(* Logix 5000 project; controller VET 1756-L62 rev 19.52; software revision 19.01; part 23 of 27 *)
(* tags used below, declared in another part *)
   Aux : DINT[500];
   Eqp : Equipo[50];
   I : Index;
   PID : PID_Struct;
   RunHours : DINT[1000];
   RunSegs : DINT[1000];
   RunStarts : DINT[1000];
   _Eqp : Equipo[800];
   _Eqp_Cfg : Eqp_Cfg[800];
   _SS : Soft_Starter[20];
   _Typlgie : Eqp_Typologie[800];   // Process Flow Typologie
   borrar : DINT[100];
   comandos : DINT[10];
   corriente : REAL[40];
   DRT : DRTs[10];
   SetDInt : DINT[500];
   simulacion : BOOL;
   SSvar : set_variables;
   Timer : TIMER[500];
(* Main1, continued *)

ROUTINE _Cntrl_Bin   (* ladder *)
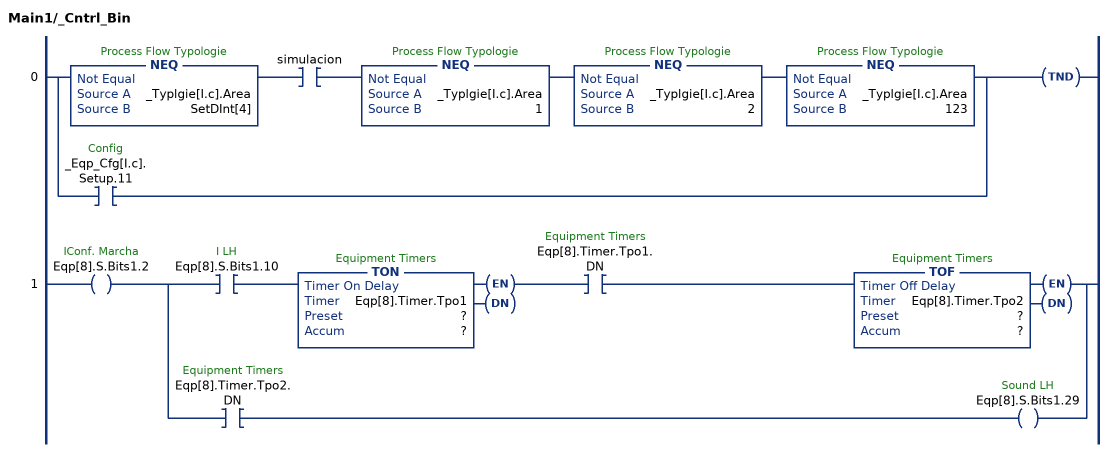
   0: [NEQ(_Typlgie[I.c].Area,SetDInt[4]) XIC(simulacion) NEQ(_Typlgie[I.c].Area,1) NEQ(_Typlgie[I.c].Area,2) NEQ(_Typlgie[I.c].Area,123) ,XIC(_Eqp_Cfg[I.c].Setup.11) ]TND();
   1: OTE(Eqp[8].S.Bits1.2)[XIC(Eqp[8].S.Bits1.10) TON(Eqp[8].Timer.Tpo1,?,?) XIC(Eqp[8].Timer.Tpo1.DN) TOF(Eqp[8].Timer.Tpo2,?,?) ,XIC(Eqp[8].Timer.Tpo2.DN) OTE(Eqp[8].S.Bits1.29) ];
END_ROUTINE

ROUTINE _Cntrl_Drot   (* ladder *)
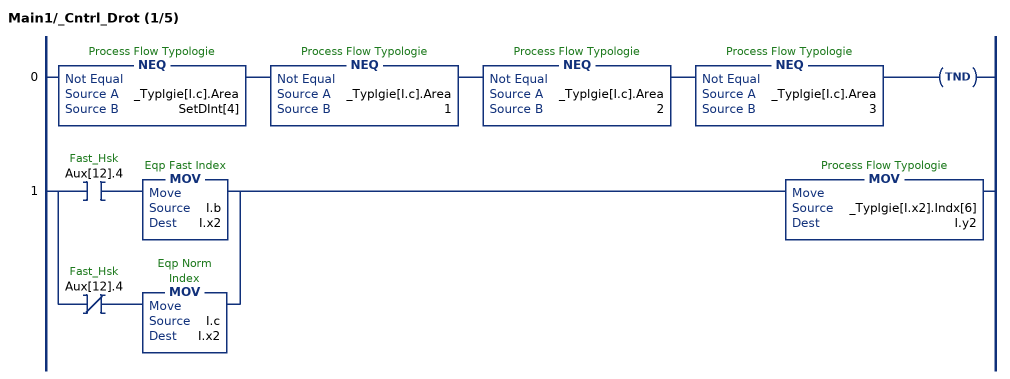
   0: NEQ(_Typlgie[I.c].Area,SetDInt[4])NEQ(_Typlgie[I.c].Area,1)NEQ(_Typlgie[I.c].Area,2)NEQ(_Typlgie[I.c].Area,3)TND();
   1: [XIC(Aux[12].4) MOV(I.b,I.x2) ,XIO(Aux[12].4) MOV(I.c,I.x2) ]MOV(_Typlgie[I.x2].Indx[6],I.y2);
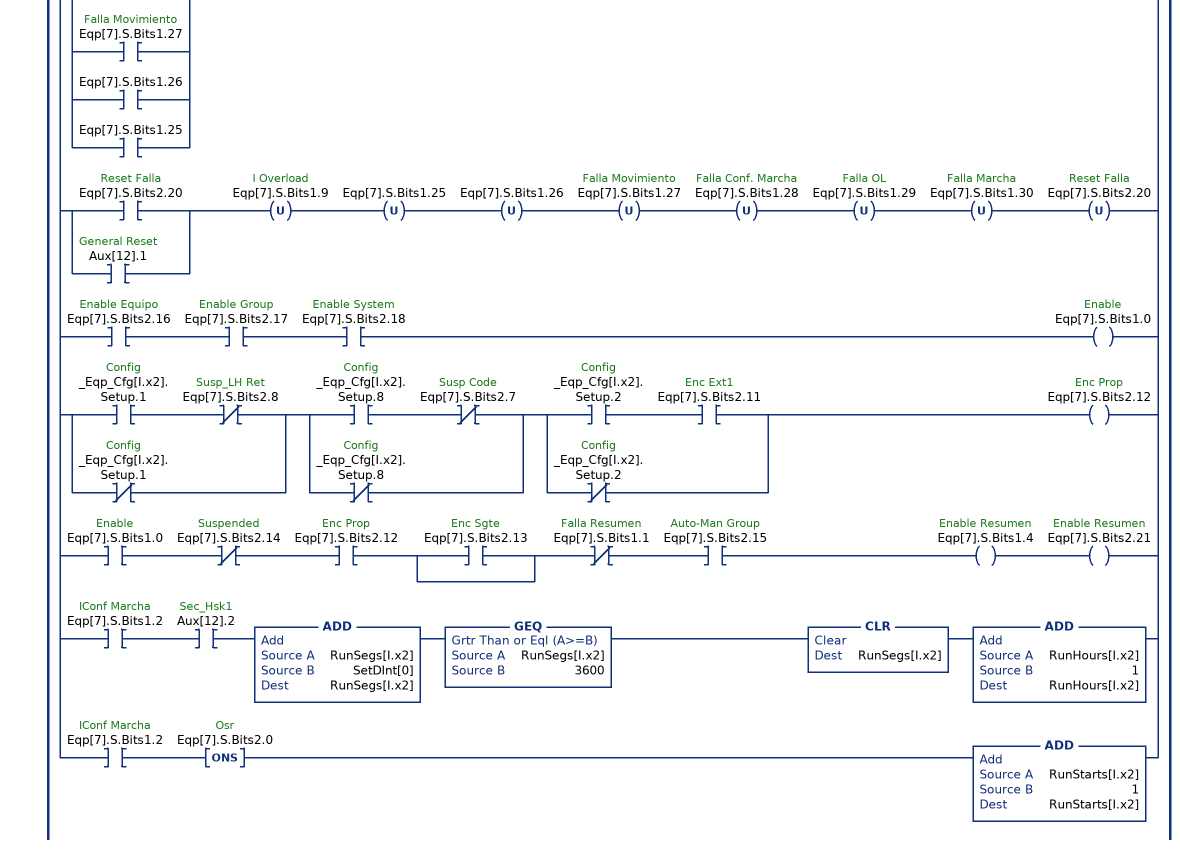
   2: [[XIC(Eqp[7].S.Bits2.31) ,XIC(_Eqp_Cfg[I.x2].Setup.14) XIC(Eqp[7].S.Bits2.30) ] XIO(Eqp[7].S.Bits1.2) XIO(Eqp[7].S.Bits1.30) TON(Eqp[7].Timer.Tpo1,?,?) XIC(Eqp[7].Timer.Tpo1.DN) OTL(Eqp[7].S.Bits1.30) ,XIC(Eqp[7].S.Bits1.9) OTL(Eqp[7].S.Bits1.29) ,TON(Eqp[7].Timer.Tpo4,?,?) XIC(Eqp[7].Timer.Tpo4.DN) OTL(Eqp[7].S.Bits1.27) ,[XIC(Eqp[7].S.Bits2.31) ,XIC(_Eqp_Cfg[I.x2].Setup.14) XIC(Eqp[7].S.Bits2.30) ] NEQ(DRT[I.y2].ConfPos,DRT[I.y2].CmdPos) TON(Eqp[7].Timer.Tpo2,?,?) XIC(Eqp[7].Timer.Tpo2.DN) OTL(Eqp[7].S.Bits1.28) ,[[XIC(Eqp[7].S.Bits2.29) XIO(Eqp[7].S.Bits1.15) ,XIO(Eqp[7].S.Bits2.29) XIO(Eqp[7].S.Bits1.14) ] ,XIO(Eqp[7].S.Bits1.14) XIO(Eqp[7].S.Bits1.15) ] TON(Eqp[7].Timer.Tpo3,?,?) ,XIC(Eqp[7].Timer.Tpo3.DN) OTL(Eqp[7].S.Bits1.26) ,XIC(Eqp[7].S.Bits1.8) TON(Eqp[7].Timer.Tpo5,?,?) XIC(Eqp[7].Timer.Tpo5.DN) OTL(Eqp[7].S.Bits1.25) ,[XIC(Eqp[7].S.Bits1.28) ,XIC(Eqp[7].S.Bits1.29) ,XIC(Eqp[7].S.Bits1.30) ,XIC(Eqp[7].S.Bits1.27) ,XIC(Eqp[7].S.Bits1.26) ,XIC(Eqp[7].S.Bits1.25) ] RES(Eqp[7].Timer.Tpo1) RES(Eqp[7].Timer.Tpo2) RES(Eqp[7].Timer.Tpo3) RES(Eqp[7].Timer.Tpo4) RES(Eqp[7].Timer.Tpo5) OTE(Eqp[7].S.Bits1.1) ,[XIC(Eqp[7].S.Bits2.20) ,XIC(Aux[12].1) ] OTU(Eqp[7].S.Bits1.9) OTU(Eqp[7].S.Bits1.25) OTU(Eqp[7].S.Bits1.26) OTU(Eqp[7].S.Bits1.27) OTU(Eqp[7].S.Bits1.28) OTU(Eqp[7].S.Bits1.29) OTU(Eqp[7].S.Bits1.30) OTU(Eqp[7].S.Bits2.20) ,XIC(Eqp[7].S.Bits2.16) XIC(Eqp[7].S.Bits2.17) XIC(Eqp[7].S.Bits2.18) OTE(Eqp[7].S.Bits1.0) ,[XIC(_Eqp_Cfg[I.x2].Setup.1) XIO(Eqp[7].S.Bits2.8) ,XIO(_Eqp_Cfg[I.x2].Setup.1) ] [XIC(_Eqp_Cfg[I.x2].Setup.8) XIO(Eqp[7].S.Bits2.7) ,XIO(_Eqp_Cfg[I.x2].Setup.8) ] [XIC(_Eqp_Cfg[I.x2].Setup.2) XIC(Eqp[7].S.Bits2.11) ,XIO(_Eqp_Cfg[I.x2].Setup.2) ] OTE(Eqp[7].S.Bits2.12) ,XIC(Eqp[7].S.Bits1.0) XIO(Eqp[7].S.Bits2.14) XIC(Eqp[7].S.Bits2.12) [XIC(Eqp[7].S.Bits2.13) ,] XIO(Eqp[7].S.Bits1.1) XIC(Eqp[7].S.Bits2.15) OTE(Eqp[7].S.Bits1.4) OTE(Eqp[7].S.Bits2.21) ,XIC(Eqp[7].S.Bits1.2) XIC(Aux[12].2) ADD(RunSegs[I.x2],SetDInt[0],RunSegs[I.x2]) GEQ(RunSegs[I.x2],3600) CLR(RunSegs[I.x2]) ADD(RunHours[I.x2],1,RunHours[I.x2]) ,XIC(Eqp[7].S.Bits1.2) ONS(Eqp[7].S.Bits2.0) ADD(RunStarts[I.x2],1,RunStarts[I.x2]) ];
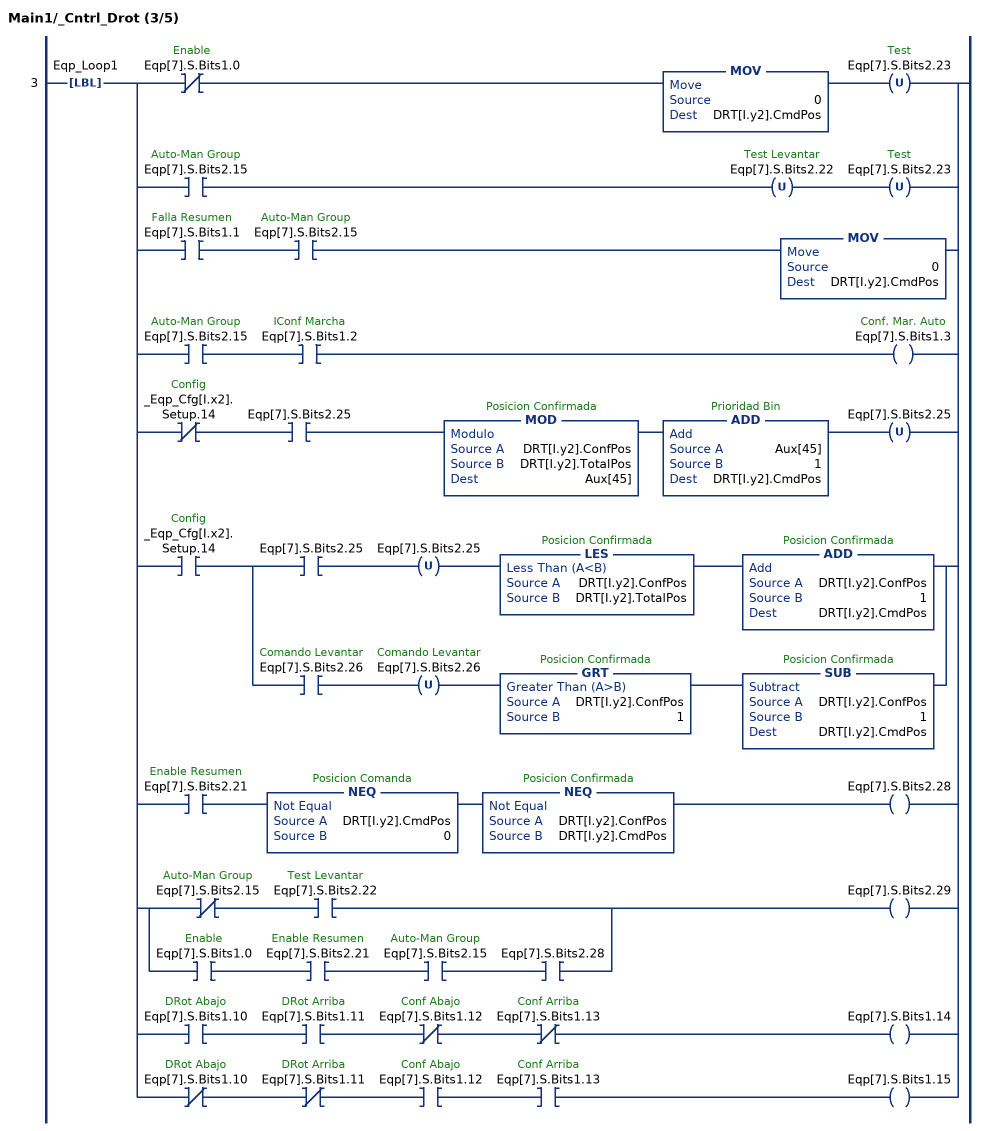
   3: LBL(Eqp_Loop1)[XIO(Eqp[7].S.Bits1.0) MOV(0,DRT[I.y2].CmdPos) OTU(Eqp[7].S.Bits2.23) ,XIC(Eqp[7].S.Bits2.15) OTU(Eqp[7].S.Bits2.22) OTU(Eqp[7].S.Bits2.23) ,XIC(Eqp[7].S.Bits1.1) XIC(Eqp[7].S.Bits2.15) MOV(0,DRT[I.y2].CmdPos) ,XIC(Eqp[7].S.Bits2.15) XIC(Eqp[7].S.Bits1.2) OTE(Eqp[7].S.Bits1.3) ,XIO(_Eqp_Cfg[I.x2].Setup.14) XIC(Eqp[7].S.Bits2.25) MOD(DRT[I.y2].ConfPos,DRT[I.y2].TotalPos,Aux[45]) ADD(Aux[45],1,DRT[I.y2].CmdPos) OTU(Eqp[7].S.Bits2.25) ,XIC(_Eqp_Cfg[I.x2].Setup.14) [XIC(Eqp[7].S.Bits2.25) OTU(Eqp[7].S.Bits2.25) LES(DRT[I.y2].ConfPos,DRT[I.y2].TotalPos) ADD(DRT[I.y2].ConfPos,1,DRT[I.y2].CmdPos) ,XIC(Eqp[7].S.Bits2.26) OTU(Eqp[7].S.Bits2.26) GRT(DRT[I.y2].ConfPos,1) SUB(DRT[I.y2].ConfPos,1,DRT[I.y2].CmdPos) ] ,XIC(Eqp[7].S.Bits2.21) NEQ(DRT[I.y2].CmdPos,0) NEQ(DRT[I.y2].ConfPos,DRT[I.y2].CmdPos) OTE(Eqp[7].S.Bits2.28) ,[XIO(Eqp[7].S.Bits2.15) XIC(Eqp[7].S.Bits2.22) ,XIC(Eqp[7].S.Bits1.0) XIC(Eqp[7].S.Bits2.21) XIC(Eqp[7].S.Bits2.15) XIC(Eqp[7].S.Bits2.28) ] OTE(Eqp[7].S.Bits2.29) ,XIC(Eqp[7].S.Bits1.10) XIC(Eqp[7].S.Bits1.11) XIO(Eqp[7].S.Bits1.12) XIO(Eqp[7].S.Bits1.13) OTE(Eqp[7].S.Bits1.14) ,XIO(Eqp[7].S.Bits1.10) XIO(Eqp[7].S.Bits1.11) XIC(Eqp[7].S.Bits1.12) XIC(Eqp[7].S.Bits1.13) OTE(Eqp[7].S.Bits1.15) ];
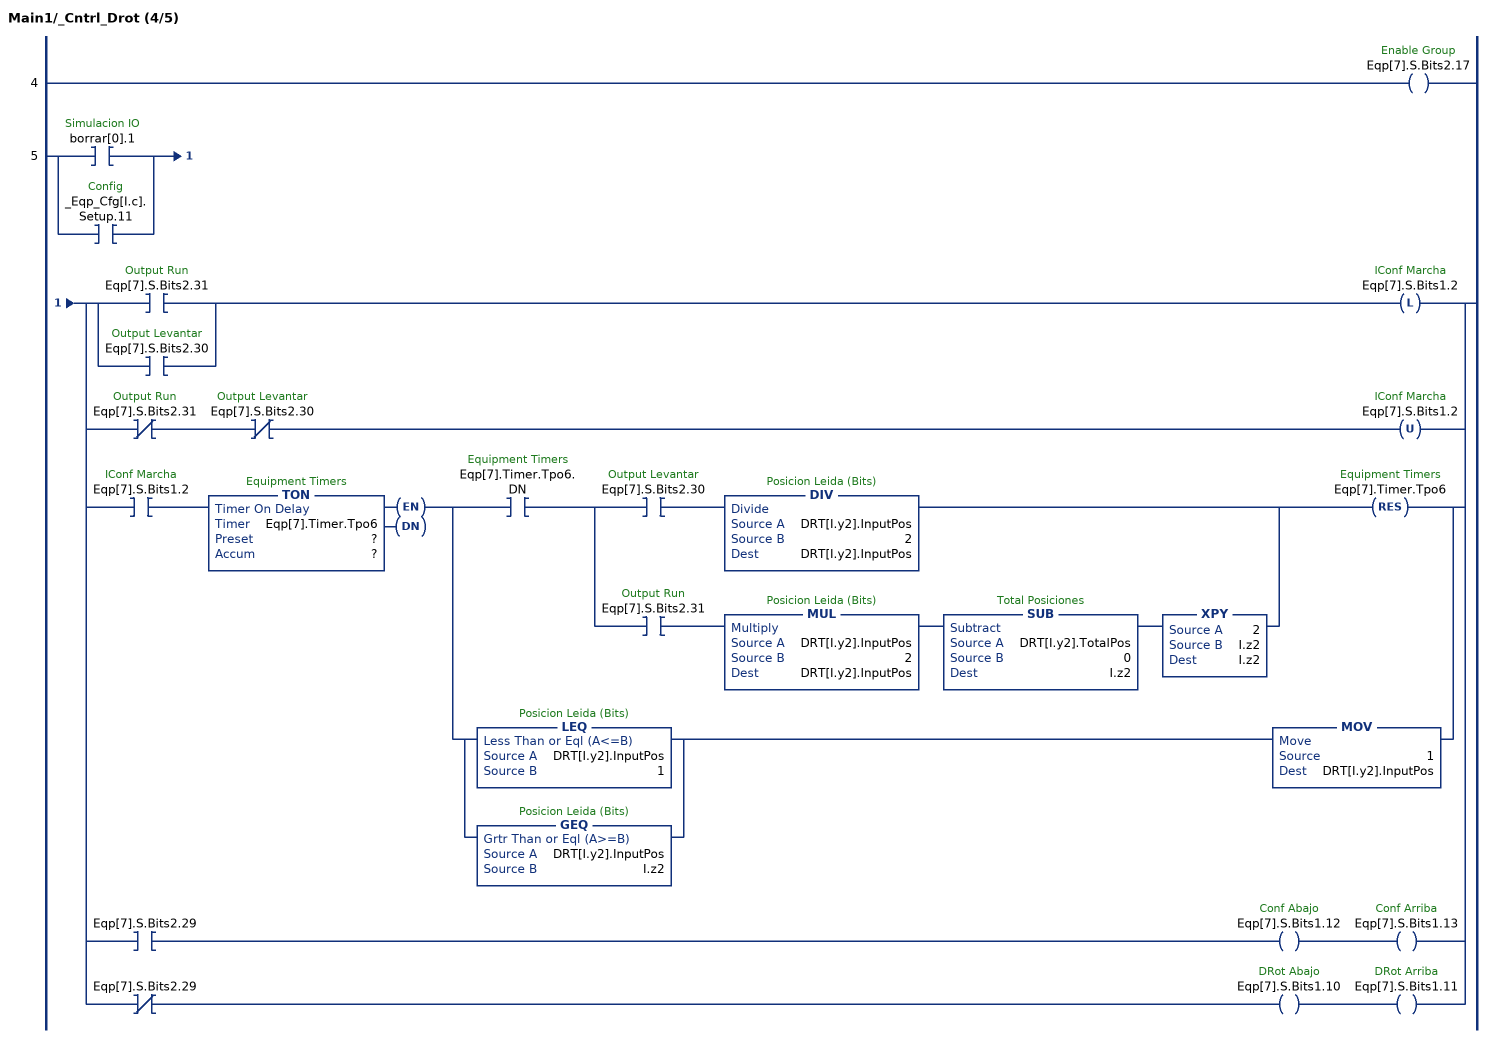
   4: OTE(Eqp[7].S.Bits2.17);
   5: [XIC(borrar[0].1) ,XIC(_Eqp_Cfg[I.c].Setup.11) ][[XIC(Eqp[7].S.Bits2.31) ,XIC(Eqp[7].S.Bits2.30) ] OTL(Eqp[7].S.Bits1.2) ,XIO(Eqp[7].S.Bits2.31) XIO(Eqp[7].S.Bits2.30) OTU(Eqp[7].S.Bits1.2) ,XIC(Eqp[7].S.Bits1.2) TON(Eqp[7].Timer.Tpo6,?,?) [XIC(Eqp[7].Timer.Tpo6.DN) [XIC(Eqp[7].S.Bits2.30) DIV(DRT[I.y2].InputPos,2,DRT[I.y2].InputPos) ,XIC(Eqp[7].S.Bits2.31) MUL(DRT[I.y2].InputPos,2,DRT[I.y2].InputPos) SUB(DRT[I.y2].TotalPos,0,I.z2) XPY(2,I.z2,I.z2) ] RES(Eqp[7].Timer.Tpo6) ,[LEQ(DRT[I.y2].InputPos,1) ,GEQ(DRT[I.y2].InputPos,I.z2) ] MOV(1,DRT[I.y2].InputPos) ] ,XIC(Eqp[7].S.Bits2.29) OTE(Eqp[7].S.Bits1.12) OTE(Eqp[7].S.Bits1.13) ,XIO(Eqp[7].S.Bits2.29) OTE(Eqp[7].S.Bits1.10) OTE(Eqp[7].S.Bits1.11) ];
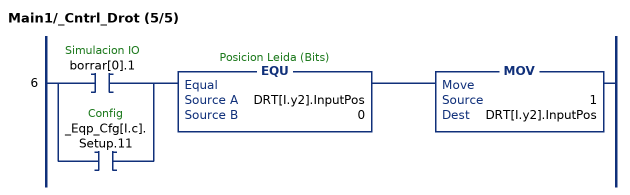
   6: [XIC(borrar[0].1) ,XIC(_Eqp_Cfg[I.c].Setup.11) ]EQU(DRT[I.y2].InputPos,0)MOV(1,DRT[I.y2].InputPos);
END_ROUTINE

ROUTINE _Cntrl_Gate   (* ladder *)
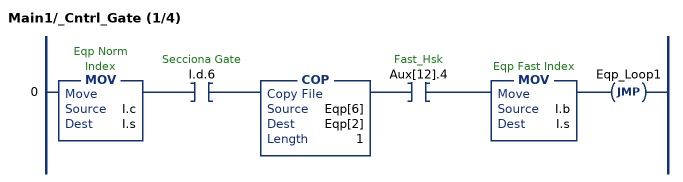
   0: MOV(I.c,I.s)XIC(I.d.6)COP(Eqp[6],Eqp[2],1)XIC(Aux[12].4)MOV(I.b,I.s)JMP(Eqp_Loop1);
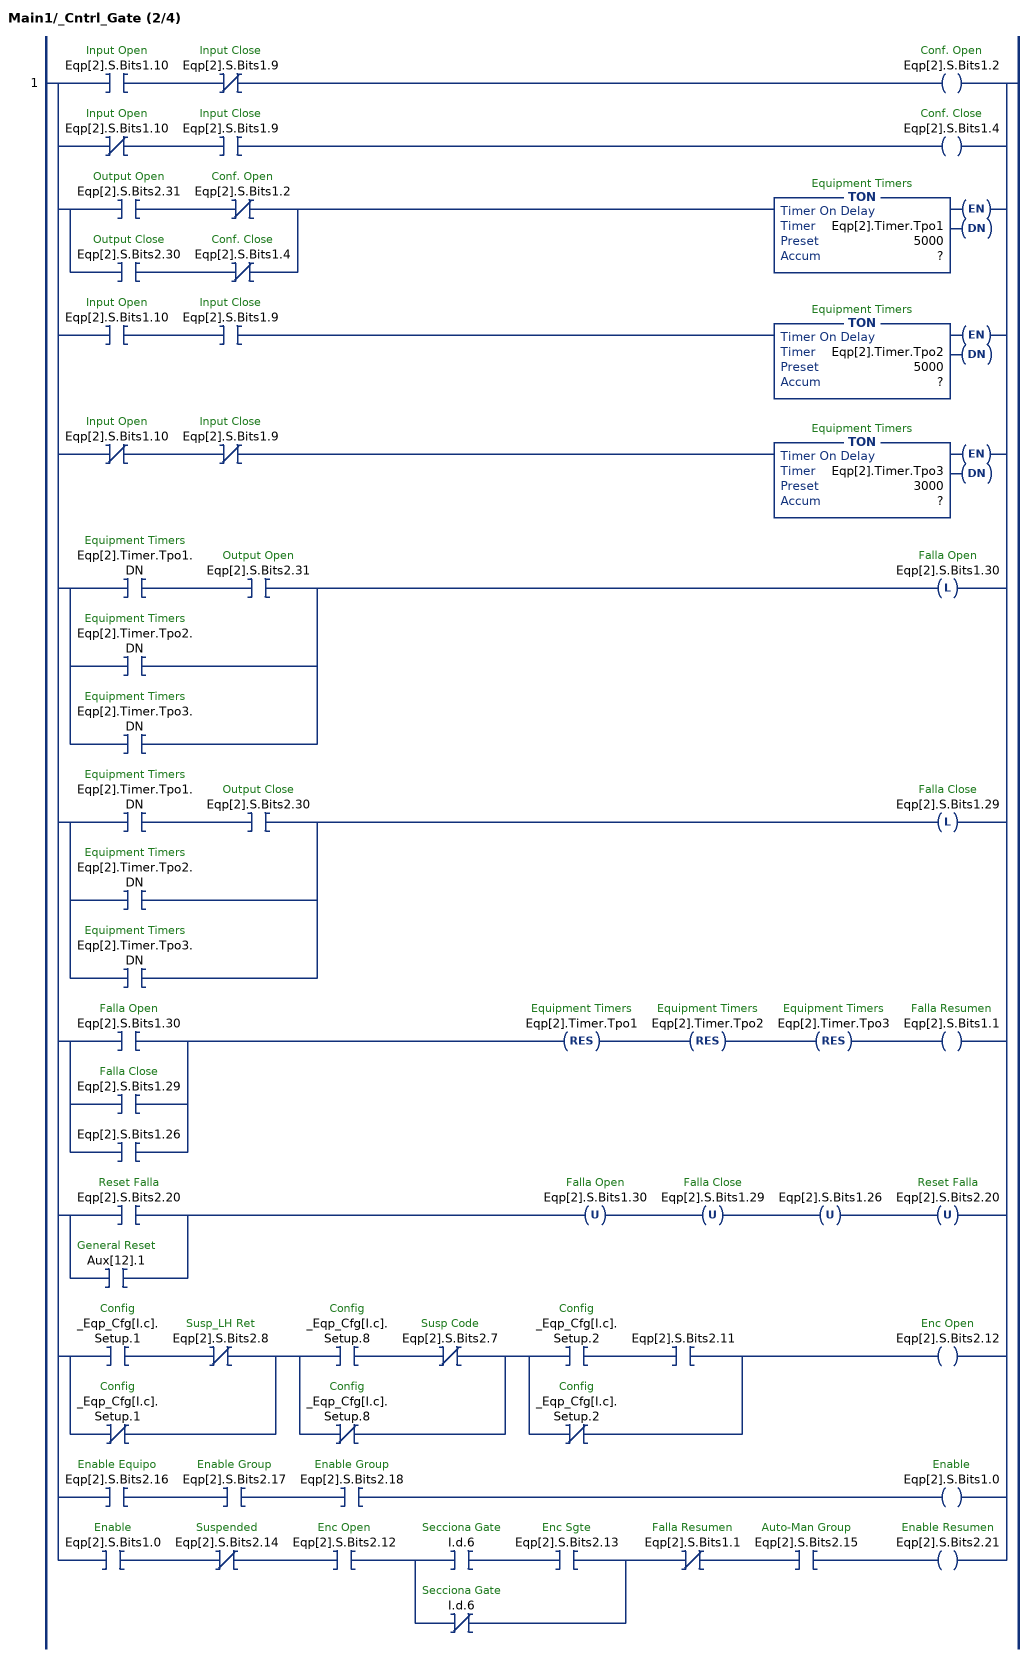
   1: [[XIC(Eqp[2].S.Bits1.10) XIO(Eqp[2].S.Bits1.9) OTE(Eqp[2].S.Bits1.2) ,XIO(Eqp[2].S.Bits1.10) XIC(Eqp[2].S.Bits1.9) OTE(Eqp[2].S.Bits1.4) ] ,[XIC(Eqp[2].S.Bits2.31) XIO(Eqp[2].S.Bits1.2) ,XIC(Eqp[2].S.Bits2.30) XIO(Eqp[2].S.Bits1.4) ] TON(Eqp[2].Timer.Tpo1,?,?) ,XIC(Eqp[2].S.Bits1.10) XIC(Eqp[2].S.Bits1.9) TON(Eqp[2].Timer.Tpo2,?,?) ,XIO(Eqp[2].S.Bits1.10) XIO(Eqp[2].S.Bits1.9) TON(Eqp[2].Timer.Tpo3,?,?) ,[XIC(Eqp[2].Timer.Tpo1.DN) XIC(Eqp[2].S.Bits2.31) ,XIC(Eqp[2].Timer.Tpo2.DN) ,XIC(Eqp[2].Timer.Tpo3.DN) ] OTL(Eqp[2].S.Bits1.30) ,[XIC(Eqp[2].Timer.Tpo1.DN) XIC(Eqp[2].S.Bits2.30) ,XIC(Eqp[2].Timer.Tpo2.DN) ,XIC(Eqp[2].Timer.Tpo3.DN) ] OTL(Eqp[2].S.Bits1.29) ,[XIC(Eqp[2].S.Bits1.30) ,XIC(Eqp[2].S.Bits1.29) ,XIC(Eqp[2].S.Bits1.26) ] RES(Eqp[2].Timer.Tpo1) RES(Eqp[2].Timer.Tpo2) RES(Eqp[2].Timer.Tpo3) OTE(Eqp[2].S.Bits1.1) ,[XIC(Eqp[2].S.Bits2.20) ,XIC(Aux[12].1) ] OTU(Eqp[2].S.Bits1.30) OTU(Eqp[2].S.Bits1.29) OTU(Eqp[2].S.Bits1.26) OTU(Eqp[2].S.Bits2.20) ,[XIC(_Eqp_Cfg[I.c].Setup.1) XIO(Eqp[2].S.Bits2.8) ,XIO(_Eqp_Cfg[I.c].Setup.1) ] [XIC(_Eqp_Cfg[I.c].Setup.8) XIO(Eqp[2].S.Bits2.7) ,XIO(_Eqp_Cfg[I.c].Setup.8) ] [XIC(_Eqp_Cfg[I.c].Setup.2) XIC(Eqp[2].S.Bits2.11) ,XIO(_Eqp_Cfg[I.c].Setup.2) ] OTE(Eqp[2].S.Bits2.12) ,XIC(Eqp[2].S.Bits2.16) XIC(Eqp[2].S.Bits2.17) XIC(Eqp[2].S.Bits2.18) OTE(Eqp[2].S.Bits1.0) ,XIC(Eqp[2].S.Bits1.0) XIO(Eqp[2].S.Bits2.14) XIC(Eqp[2].S.Bits2.12) [XIC(I.d.6) XIC(Eqp[2].S.Bits2.13) ,XIO(I.d.6) ] XIO(Eqp[2].S.Bits1.1) XIC(Eqp[2].S.Bits2.15) OTE(Eqp[2].S.Bits2.21) ];
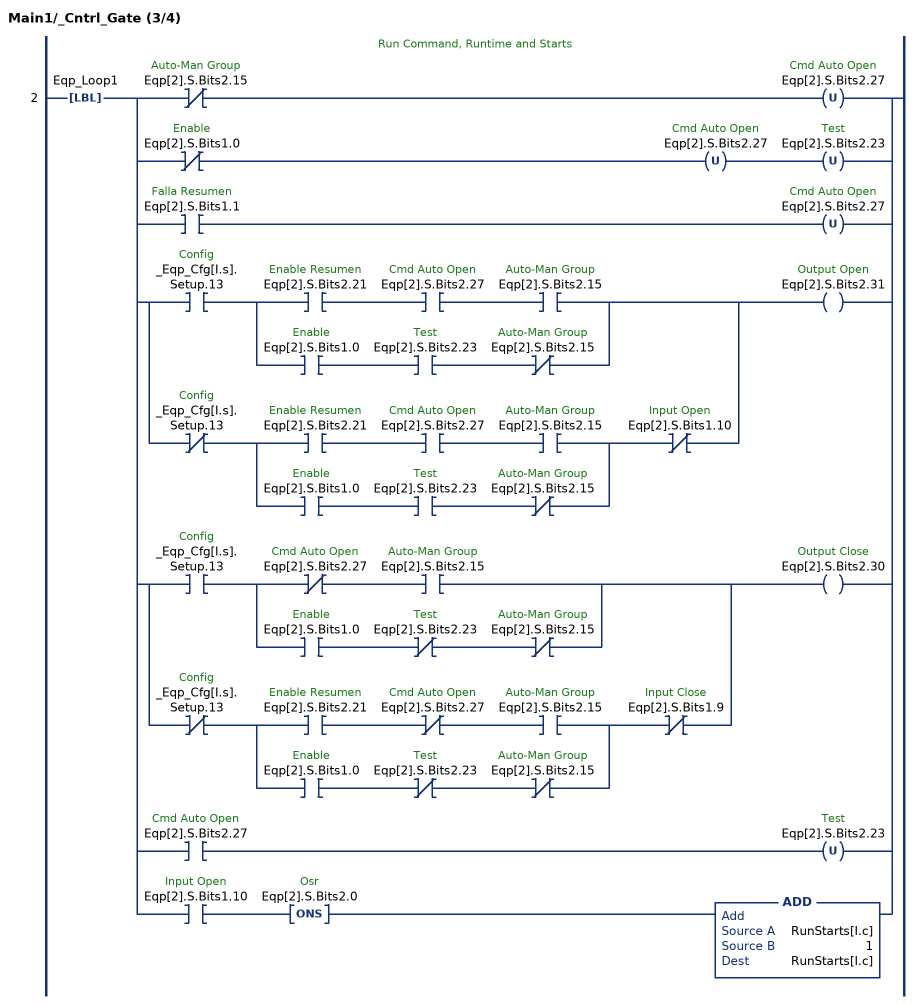
   // Run Command, Runtime and Starts
   2: LBL(Eqp_Loop1)[XIO(Eqp[2].S.Bits2.15) OTU(Eqp[2].S.Bits2.27) ,XIO(Eqp[2].S.Bits1.0) OTU(Eqp[2].S.Bits2.27) OTU(Eqp[2].S.Bits2.23) ,XIC(Eqp[2].S.Bits1.1) OTU(Eqp[2].S.Bits2.27) ,[XIC(_Eqp_Cfg[I.s].Setup.13) [XIC(Eqp[2].S.Bits2.21) XIC(Eqp[2].S.Bits2.27) XIC(Eqp[2].S.Bits2.15) ,XIC(Eqp[2].S.Bits1.0) XIC(Eqp[2].S.Bits2.23) XIO(Eqp[2].S.Bits2.15) ] ,XIO(_Eqp_Cfg[I.s].Setup.13) [XIC(Eqp[2].S.Bits2.21) XIC(Eqp[2].S.Bits2.27) XIC(Eqp[2].S.Bits2.15) ,XIC(Eqp[2].S.Bits1.0) XIC(Eqp[2].S.Bits2.23) XIO(Eqp[2].S.Bits2.15) ] XIO(Eqp[2].S.Bits1.10) ] OTE(Eqp[2].S.Bits2.31) ,[XIC(_Eqp_Cfg[I.s].Setup.13) [XIO(Eqp[2].S.Bits2.27) XIC(Eqp[2].S.Bits2.15) ,XIC(Eqp[2].S.Bits1.0) XIO(Eqp[2].S.Bits2.23) XIO(Eqp[2].S.Bits2.15) ] ,XIO(_Eqp_Cfg[I.s].Setup.13) [XIC(Eqp[2].S.Bits2.21) XIO(Eqp[2].S.Bits2.27) XIC(Eqp[2].S.Bits2.15) ,XIC(Eqp[2].S.Bits1.0) XIO(Eqp[2].S.Bits2.23) XIO(Eqp[2].S.Bits2.15) ] XIO(Eqp[2].S.Bits1.9) ] OTE(Eqp[2].S.Bits2.30) ,XIC(Eqp[2].S.Bits2.27) OTU(Eqp[2].S.Bits2.23) ,XIC(Eqp[2].S.Bits1.10) ONS(Eqp[2].S.Bits2.0) ADD(RunStarts[I.c],1,RunStarts[I.c]) ];
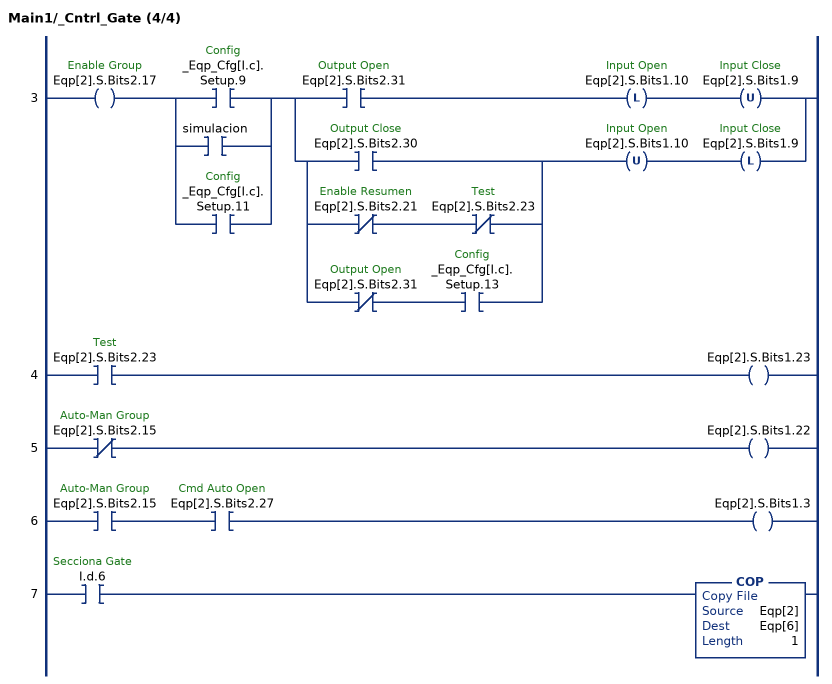
   3: OTE(Eqp[2].S.Bits2.17)[XIC(_Eqp_Cfg[I.c].Setup.9) ,XIC(simulacion) ,XIC(_Eqp_Cfg[I.c].Setup.11) ][XIC(Eqp[2].S.Bits2.31) OTL(Eqp[2].S.Bits1.10) OTU(Eqp[2].S.Bits1.9) ,[XIC(Eqp[2].S.Bits2.30) ,XIO(Eqp[2].S.Bits2.21) XIO(Eqp[2].S.Bits2.23) ,XIO(Eqp[2].S.Bits2.31) XIC(_Eqp_Cfg[I.c].Setup.13) ] OTU(Eqp[2].S.Bits1.10) OTL(Eqp[2].S.Bits1.9) ];
   4: XIC(Eqp[2].S.Bits2.23)OTE(Eqp[2].S.Bits1.23);
   5: XIO(Eqp[2].S.Bits2.15)OTE(Eqp[2].S.Bits1.22);
   6: XIC(Eqp[2].S.Bits2.15)XIC(Eqp[2].S.Bits2.27)OTE(Eqp[2].S.Bits1.3);
   7: XIC(I.d.6)COP(Eqp[2],Eqp[6],1);
END_ROUTINE

ROUTINE _Cntrl_Motor   (* ladder *)
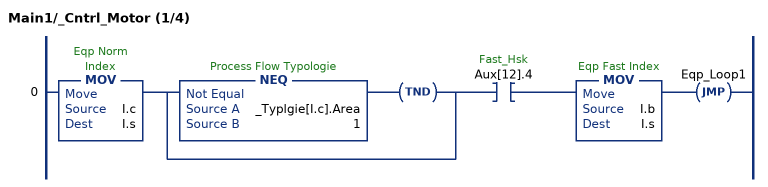
   0: MOV(I.c,I.s)[NEQ(_Typlgie[I.c].Area,1) TND() ,]XIC(Aux[12].4)MOV(I.b,I.s)JMP(Eqp_Loop1);
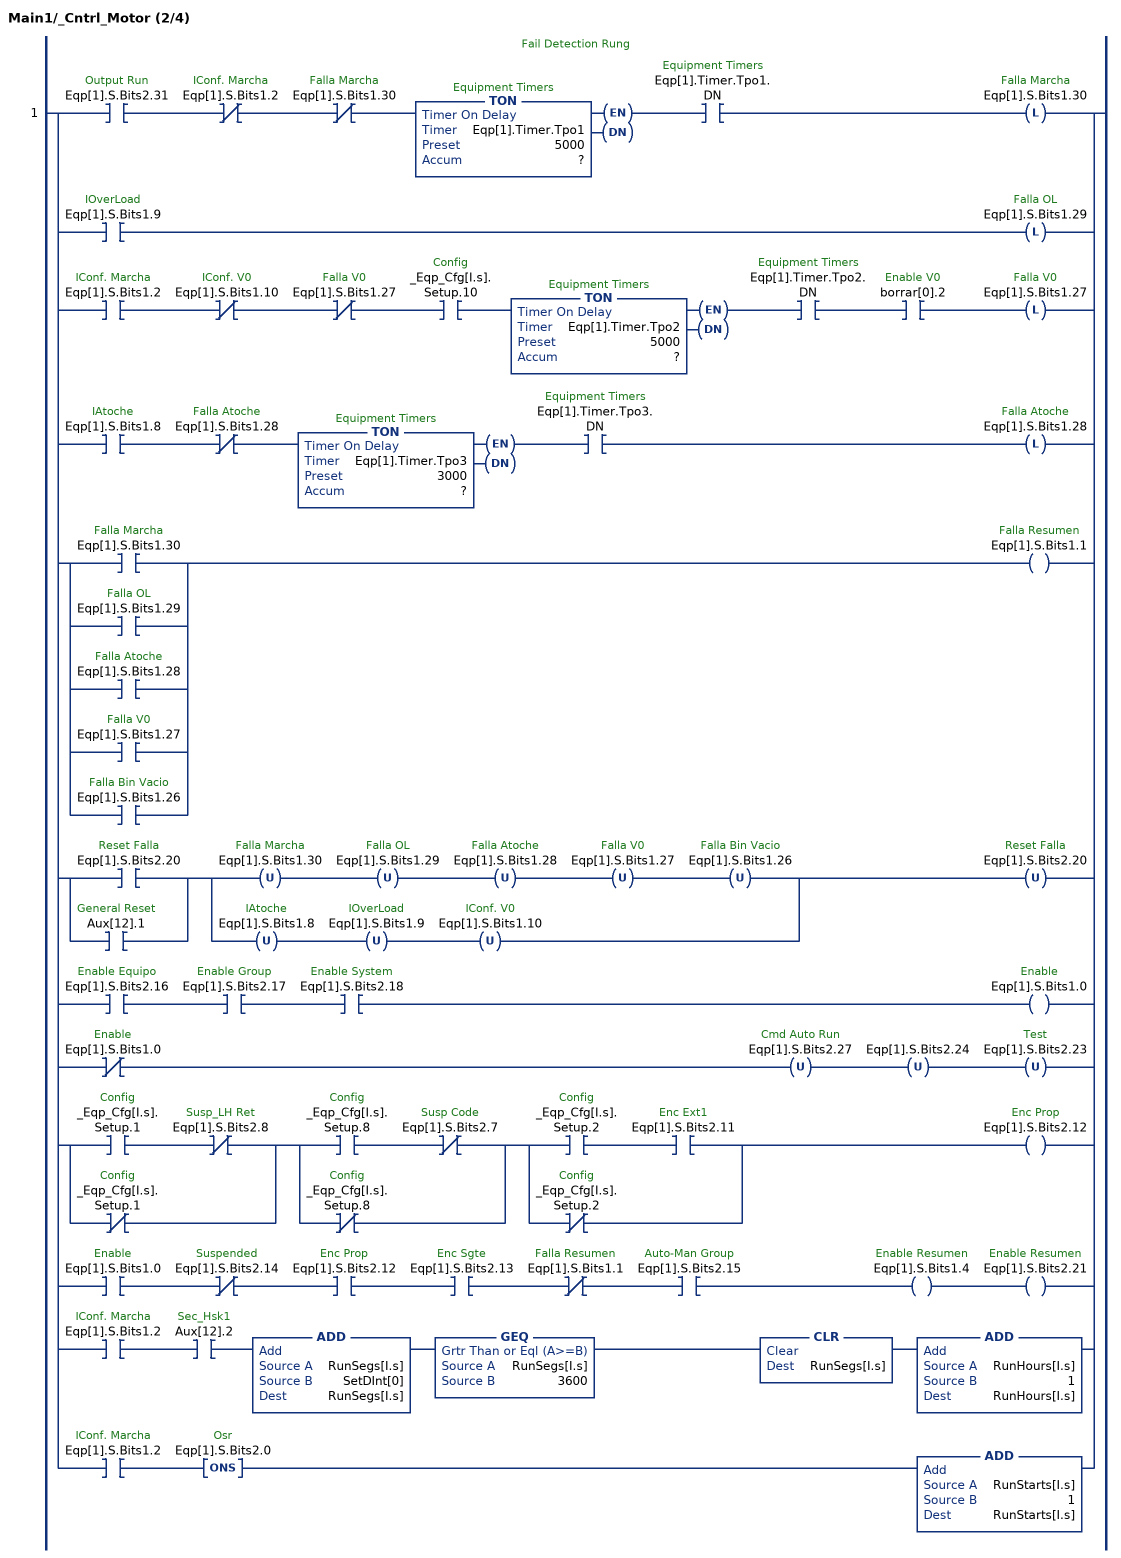
   // Fail Detection Rung
   1: [XIC(Eqp[1].S.Bits2.31) XIO(Eqp[1].S.Bits1.2) XIO(Eqp[1].S.Bits1.30) TON(Eqp[1].Timer.Tpo1,?,?) XIC(Eqp[1].Timer.Tpo1.DN) OTL(Eqp[1].S.Bits1.30) ,XIC(Eqp[1].S.Bits1.9) OTL(Eqp[1].S.Bits1.29) ,XIC(Eqp[1].S.Bits1.2) XIO(Eqp[1].S.Bits1.10) XIO(Eqp[1].S.Bits1.27) XIC(_Eqp_Cfg[I.s].Setup.10) TON(Eqp[1].Timer.Tpo2,?,?) XIC(Eqp[1].Timer.Tpo2.DN) XIC(borrar[0].2) OTL(Eqp[1].S.Bits1.27) ,XIC(Eqp[1].S.Bits1.8) XIO(Eqp[1].S.Bits1.28) TON(Eqp[1].Timer.Tpo3,?,?) XIC(Eqp[1].Timer.Tpo3.DN) OTL(Eqp[1].S.Bits1.28) ,[XIC(Eqp[1].S.Bits1.30) ,XIC(Eqp[1].S.Bits1.29) ,XIC(Eqp[1].S.Bits1.28) ,XIC(Eqp[1].S.Bits1.27) ,XIC(Eqp[1].S.Bits1.26) ] OTE(Eqp[1].S.Bits1.1) ,[XIC(Eqp[1].S.Bits2.20) ,XIC(Aux[12].1) ] [OTU(Eqp[1].S.Bits1.30) OTU(Eqp[1].S.Bits1.29) OTU(Eqp[1].S.Bits1.28) OTU(Eqp[1].S.Bits1.27) OTU(Eqp[1].S.Bits1.26) ,OTU(Eqp[1].S.Bits1.8) OTU(Eqp[1].S.Bits1.9) OTU(Eqp[1].S.Bits1.10) ] OTU(Eqp[1].S.Bits2.20) ,[XIC(Eqp[1].S.Bits2.16) XIC(Eqp[1].S.Bits2.17) XIC(Eqp[1].S.Bits2.18) OTE(Eqp[1].S.Bits1.0) ,XIO(Eqp[1].S.Bits1.0) OTU(Eqp[1].S.Bits2.27) OTU(Eqp[1].S.Bits2.24) OTU(Eqp[1].S.Bits2.23) ] ,[XIC(_Eqp_Cfg[I.s].Setup.1) XIO(Eqp[1].S.Bits2.8) ,XIO(_Eqp_Cfg[I.s].Setup.1) ] [XIC(_Eqp_Cfg[I.s].Setup.8) XIO(Eqp[1].S.Bits2.7) ,XIO(_Eqp_Cfg[I.s].Setup.8) ] [XIC(_Eqp_Cfg[I.s].Setup.2) XIC(Eqp[1].S.Bits2.11) ,XIO(_Eqp_Cfg[I.s].Setup.2) ] OTE(Eqp[1].S.Bits2.12) ,XIC(Eqp[1].S.Bits1.0) XIO(Eqp[1].S.Bits2.14) XIC(Eqp[1].S.Bits2.12) XIC(Eqp[1].S.Bits2.13) XIO(Eqp[1].S.Bits1.1) XIC(Eqp[1].S.Bits2.15) OTE(Eqp[1].S.Bits1.4) OTE(Eqp[1].S.Bits2.21) ,XIC(Eqp[1].S.Bits1.2) XIC(Aux[12].2) ADD(RunSegs[I.s],SetDInt[0],RunSegs[I.s]) GEQ(RunSegs[I.s],3600) CLR(RunSegs[I.s]) ADD(RunHours[I.s],1,RunHours[I.s]) ,XIC(Eqp[1].S.Bits1.2) ONS(Eqp[1].S.Bits2.0) ADD(RunStarts[I.s],1,RunStarts[I.s]) ];
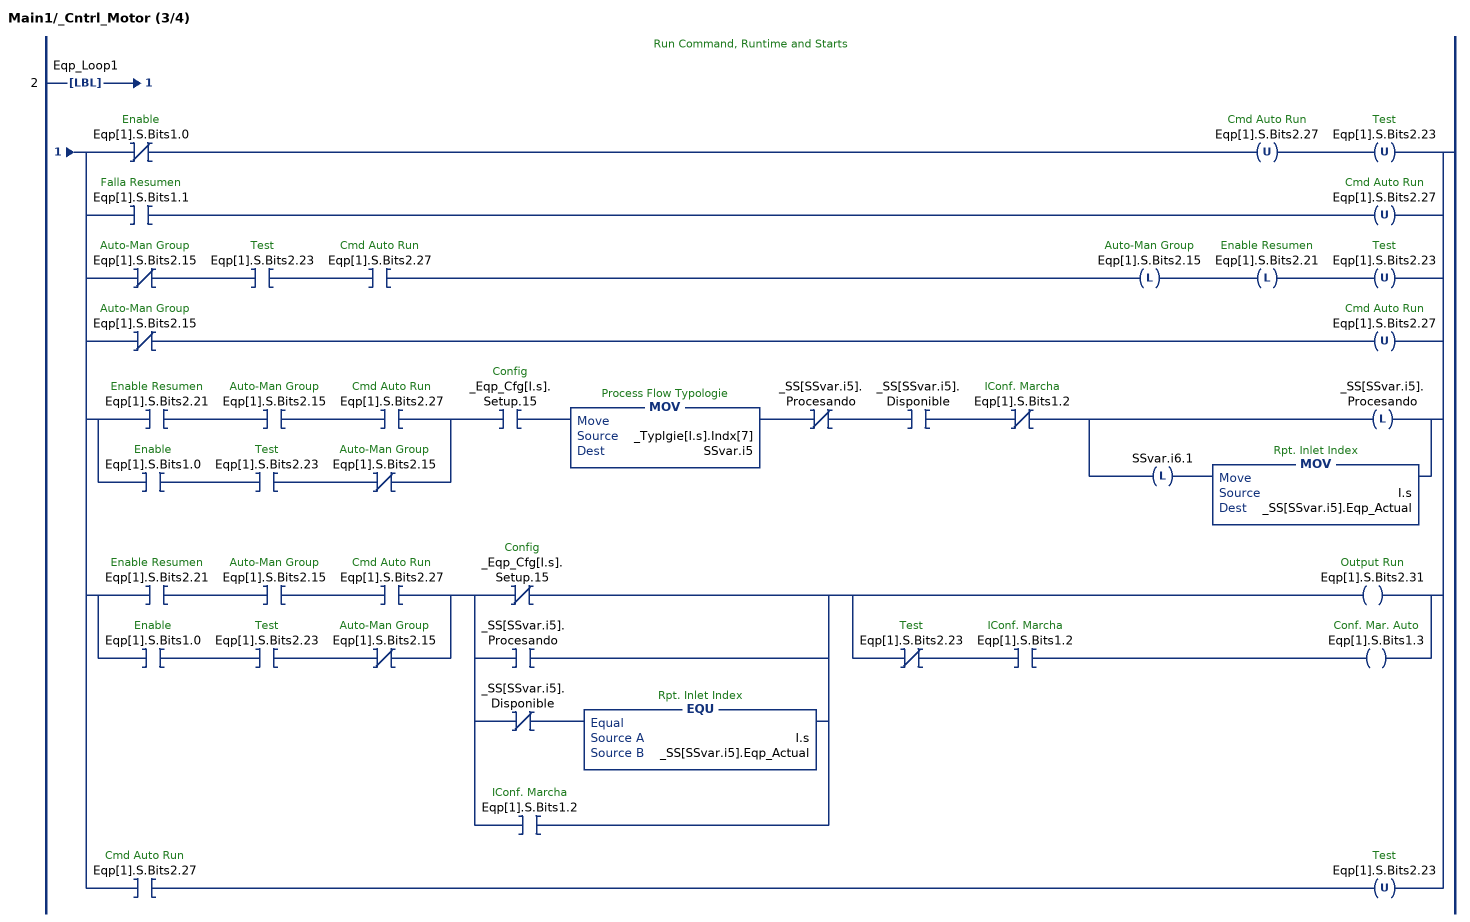
   // Run Command, Runtime and Starts
   2: LBL(Eqp_Loop1)[XIO(Eqp[1].S.Bits1.0) OTU(Eqp[1].S.Bits2.27) OTU(Eqp[1].S.Bits2.23) ,XIC(Eqp[1].S.Bits1.1) OTU(Eqp[1].S.Bits2.27) ,XIO(Eqp[1].S.Bits2.15) XIC(Eqp[1].S.Bits2.23) XIC(Eqp[1].S.Bits2.27) OTL(Eqp[1].S.Bits2.15) OTL(Eqp[1].S.Bits2.21) OTU(Eqp[1].S.Bits2.23) ,XIO(Eqp[1].S.Bits2.15) OTU(Eqp[1].S.Bits2.27) ,[XIC(Eqp[1].S.Bits2.21) XIC(Eqp[1].S.Bits2.15) XIC(Eqp[1].S.Bits2.27) ,XIC(Eqp[1].S.Bits1.0) XIC(Eqp[1].S.Bits2.23) XIO(Eqp[1].S.Bits2.15) ] XIC(_Eqp_Cfg[I.s].Setup.15) MOV(_Typlgie[I.s].Indx[7],SSvar.i5) XIO(_SS[SSvar.i5].Procesando) XIC(_SS[SSvar.i5].Disponible) XIO(Eqp[1].S.Bits1.2) [OTL(_SS[SSvar.i5].Procesando) ,OTL(SSvar.i6.1) MOV(I.s,_SS[SSvar.i5].Eqp_Actual) ] ,[XIC(Eqp[1].S.Bits2.21) XIC(Eqp[1].S.Bits2.15) XIC(Eqp[1].S.Bits2.27) ,XIC(Eqp[1].S.Bits1.0) XIC(Eqp[1].S.Bits2.23) XIO(Eqp[1].S.Bits2.15) ] [XIO(_Eqp_Cfg[I.s].Setup.15) ,[XIC(_SS[SSvar.i5].Procesando) ,XIO(_SS[SSvar.i5].Disponible) EQU(I.s,_SS[SSvar.i5].Eqp_Actual) ,XIC(Eqp[1].S.Bits1.2) ] ] [OTE(Eqp[1].S.Bits2.31) ,XIO(Eqp[1].S.Bits2.23) XIC(Eqp[1].S.Bits1.2) OTE(Eqp[1].S.Bits1.3) ] ,XIC(Eqp[1].S.Bits2.27) OTU(Eqp[1].S.Bits2.23) ];
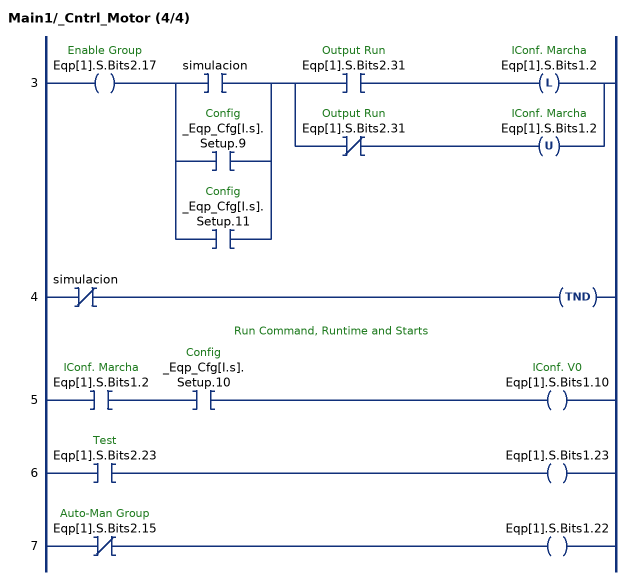
   3: OTE(Eqp[1].S.Bits2.17)[XIC(simulacion) ,XIC(_Eqp_Cfg[I.s].Setup.9) ,XIC(_Eqp_Cfg[I.s].Setup.11) ][XIC(Eqp[1].S.Bits2.31) OTL(Eqp[1].S.Bits1.2) ,XIO(Eqp[1].S.Bits2.31) OTU(Eqp[1].S.Bits1.2) ];
   4: XIO(simulacion)TND();
   // Run Command, Runtime and Starts
   5: XIC(Eqp[1].S.Bits1.2)XIC(_Eqp_Cfg[I.s].Setup.10)OTE(Eqp[1].S.Bits1.10);
   6: XIC(Eqp[1].S.Bits2.23)OTE(Eqp[1].S.Bits1.23);
   7: XIO(Eqp[1].S.Bits2.15)OTE(Eqp[1].S.Bits1.22);
END_ROUTINE

ROUTINE _Cntrl_PID   (* ladder *)
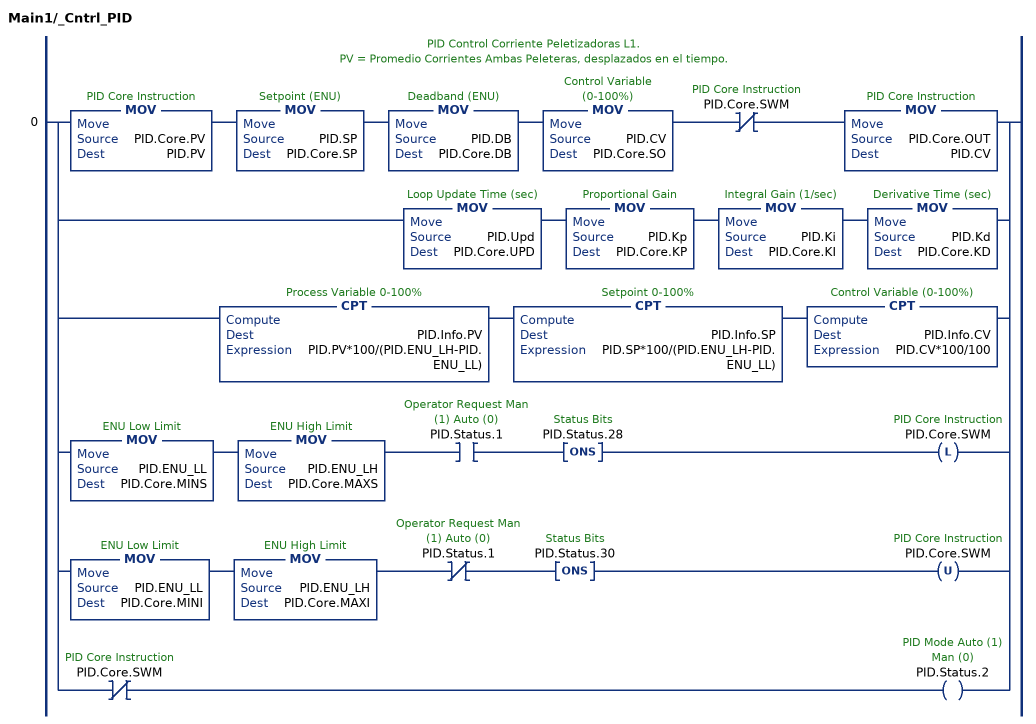
   // PID Control Corriente Peletizadoras L1.
   // PV = Promedio Corrientes Ambas Peleteras, desplazados en el tiempo.
   0: [MOV(PID.Core.PV,PID.PV) MOV(PID.SP,PID.Core.SP) MOV(PID.DB,PID.Core.DB) MOV(PID.CV,PID.Core.SO) XIO(PID.Core.SWM) MOV(PID.Core.OUT,PID.CV) ,MOV(PID.Upd,PID.Core.UPD) MOV(PID.Kp,PID.Core.KP) MOV(PID.Ki,PID.Core.KI) MOV(PID.Kd,PID.Core.KD) ,CPT(PID.Info.PV,PID.PV*100/(PID.ENU_LH-PID.ENU_LL)) CPT(PID.Info.SP,PID.SP*100/(PID.ENU_LH-PID.ENU_LL)) CPT(PID.Info.CV,PID.CV*100/100) ,MOV(PID.ENU_LL,PID.Core.MINS) MOV(PID.ENU_LH,PID.Core.MAXS) XIC(PID.Status.1) ONS(PID.Status.28) OTL(PID.Core.SWM) ,MOV(PID.ENU_LL,PID.Core.MINI) MOV(PID.ENU_LH,PID.Core.MAXI) XIO(PID.Status.1) ONS(PID.Status.30) OTU(PID.Core.SWM) ,XIO(PID.Core.SWM) OTE(PID.Status.2) ];
END_ROUTINE

ROUTINE _Cntrl_System   (* ladder *)
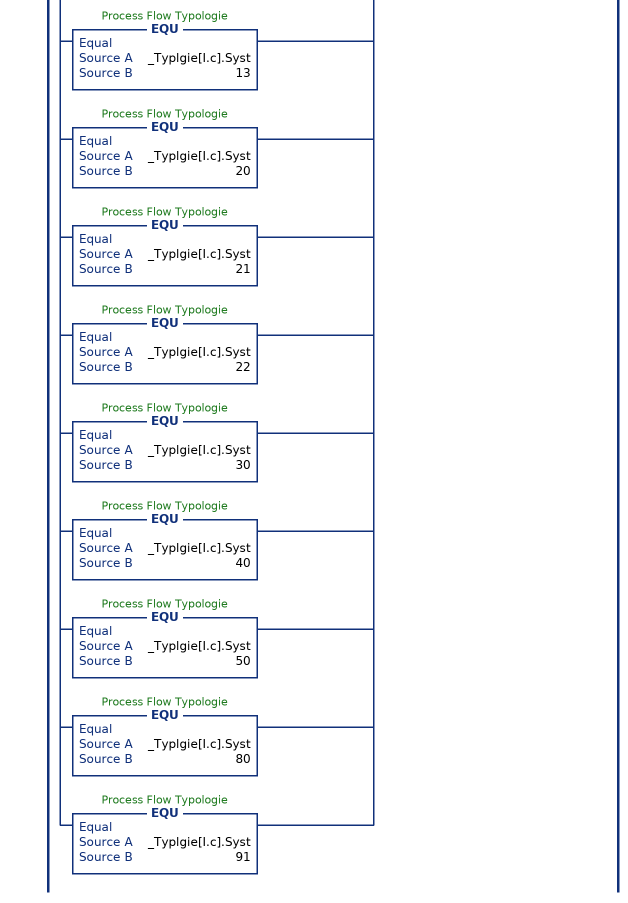
   // RSView32 General Commands
   0: [[XIC(comandos[1].0) EQU(_Typlgie[I.c].Syst,1) ,XIC(comandos[1].1) EQU(_Typlgie[I.c].Syst,2) ,XIC(comandos[1].2) EQU(_Typlgie[I.c].Syst,3) ,XIC(comandos[1].3) EQU(_Typlgie[I.c].Syst,4) ,XIC(comandos[1].4) EQU(_Typlgie[I.c].Syst,5) ,XIC(comandos[1].5) EQU(_Typlgie[I.c].Syst,6) ,XIC(comandos[1].6) EQU(_Typlgie[I.c].Syst,7) ] ,EQU(_Typlgie[I.c].Syst,10) ,[EQU(_Typlgie[I.c].Syst,11) ,EQU(_Typlgie[I.c].Syst,12) ,EQU(_Typlgie[I.c].Syst,13) ,EQU(_Typlgie[I.c].Syst,20) ,EQU(_Typlgie[I.c].Syst,21) ,EQU(_Typlgie[I.c].Syst,22) ,EQU(_Typlgie[I.c].Syst,30) ] ,EQU(_Typlgie[I.c].Syst,40) ,EQU(_Typlgie[I.c].Syst,50) ,EQU(_Typlgie[I.c].Syst,80) ,EQU(_Typlgie[I.c].Syst,91) ]OTE(_Eqp[I.c].S.Bits2.18);
END_ROUTINE

ROUTINE _Cntrl_Trifurc   (* ladder *)
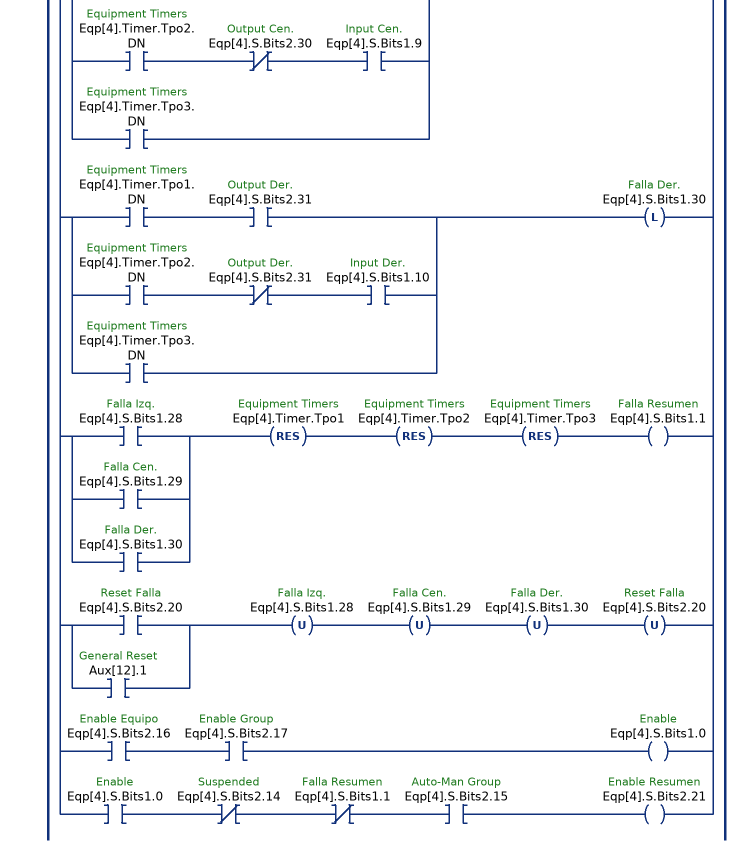
   // Fail Detection Rung
   0: [[XIC(Eqp[4].S.Bits1.8) XIO(Eqp[4].S.Bits1.9) XIO(Eqp[4].S.Bits1.10) OTE(Eqp[4].S.Bits1.2) ,XIO(Eqp[4].S.Bits1.8) XIC(Eqp[4].S.Bits1.9) XIO(Eqp[4].S.Bits1.10) OTE(Eqp[4].S.Bits1.3) ,XIO(Eqp[4].S.Bits1.8) XIO(Eqp[4].S.Bits1.9) XIC(Eqp[4].S.Bits1.10) OTE(Eqp[4].S.Bits1.4) ] ,[XIC(Eqp[4].S.Bits2.29) XIO(Eqp[4].S.Bits1.2) ,XIC(Eqp[4].S.Bits2.30) XIO(Eqp[4].S.Bits1.3) ,XIC(Eqp[4].S.Bits2.31) XIO(Eqp[4].S.Bits1.4) ] TON(Eqp[4].Timer.Tpo1,?,?) ,[XIC(Eqp[4].S.Bits1.8) XIC(Eqp[4].S.Bits1.9) ,XIC(Eqp[4].S.Bits1.8) XIC(Eqp[4].S.Bits1.10) ,XIC(Eqp[4].S.Bits1.9) XIC(Eqp[4].S.Bits1.10) ] TON(Eqp[4].Timer.Tpo2,?,?) ,XIO(Eqp[4].S.Bits1.8) XIO(Eqp[4].S.Bits1.9) XIO(Eqp[4].S.Bits1.10) TON(Eqp[4].Timer.Tpo3,?,?) ,[XIC(Eqp[4].Timer.Tpo1.DN) XIC(Eqp[4].S.Bits2.29) ,XIC(Eqp[4].Timer.Tpo2.DN) XIO(Eqp[4].S.Bits2.29) XIC(Eqp[4].S.Bits1.8) ,XIC(Eqp[4].Timer.Tpo3.DN) ] OTL(Eqp[4].S.Bits1.28) ,[XIC(Eqp[4].Timer.Tpo1.DN) XIC(Eqp[4].S.Bits2.30) ,XIC(Eqp[4].Timer.Tpo2.DN) XIO(Eqp[4].S.Bits2.30) XIC(Eqp[4].S.Bits1.9) ,XIC(Eqp[4].Timer.Tpo3.DN) ] OTL(Eqp[4].S.Bits1.29) ,[XIC(Eqp[4].Timer.Tpo1.DN) XIC(Eqp[4].S.Bits2.31) ,XIC(Eqp[4].Timer.Tpo2.DN) XIO(Eqp[4].S.Bits2.31) XIC(Eqp[4].S.Bits1.10) ,XIC(Eqp[4].Timer.Tpo3.DN) ] OTL(Eqp[4].S.Bits1.30) ,[XIC(Eqp[4].S.Bits1.28) ,XIC(Eqp[4].S.Bits1.29) ,XIC(Eqp[4].S.Bits1.30) ] RES(Eqp[4].Timer.Tpo1) RES(Eqp[4].Timer.Tpo2) RES(Eqp[4].Timer.Tpo3) OTE(Eqp[4].S.Bits1.1) ,[XIC(Eqp[4].S.Bits2.20) ,XIC(Aux[12].1) ] OTU(Eqp[4].S.Bits1.28) OTU(Eqp[4].S.Bits1.29) OTU(Eqp[4].S.Bits1.30) OTU(Eqp[4].S.Bits2.20) ,XIC(Eqp[4].S.Bits2.16) XIC(Eqp[4].S.Bits2.17) OTE(Eqp[4].S.Bits1.0) ,XIC(Eqp[4].S.Bits1.0) XIO(Eqp[4].S.Bits2.14) XIO(Eqp[4].S.Bits1.1) XIC(Eqp[4].S.Bits2.15) OTE(Eqp[4].S.Bits2.21) ];
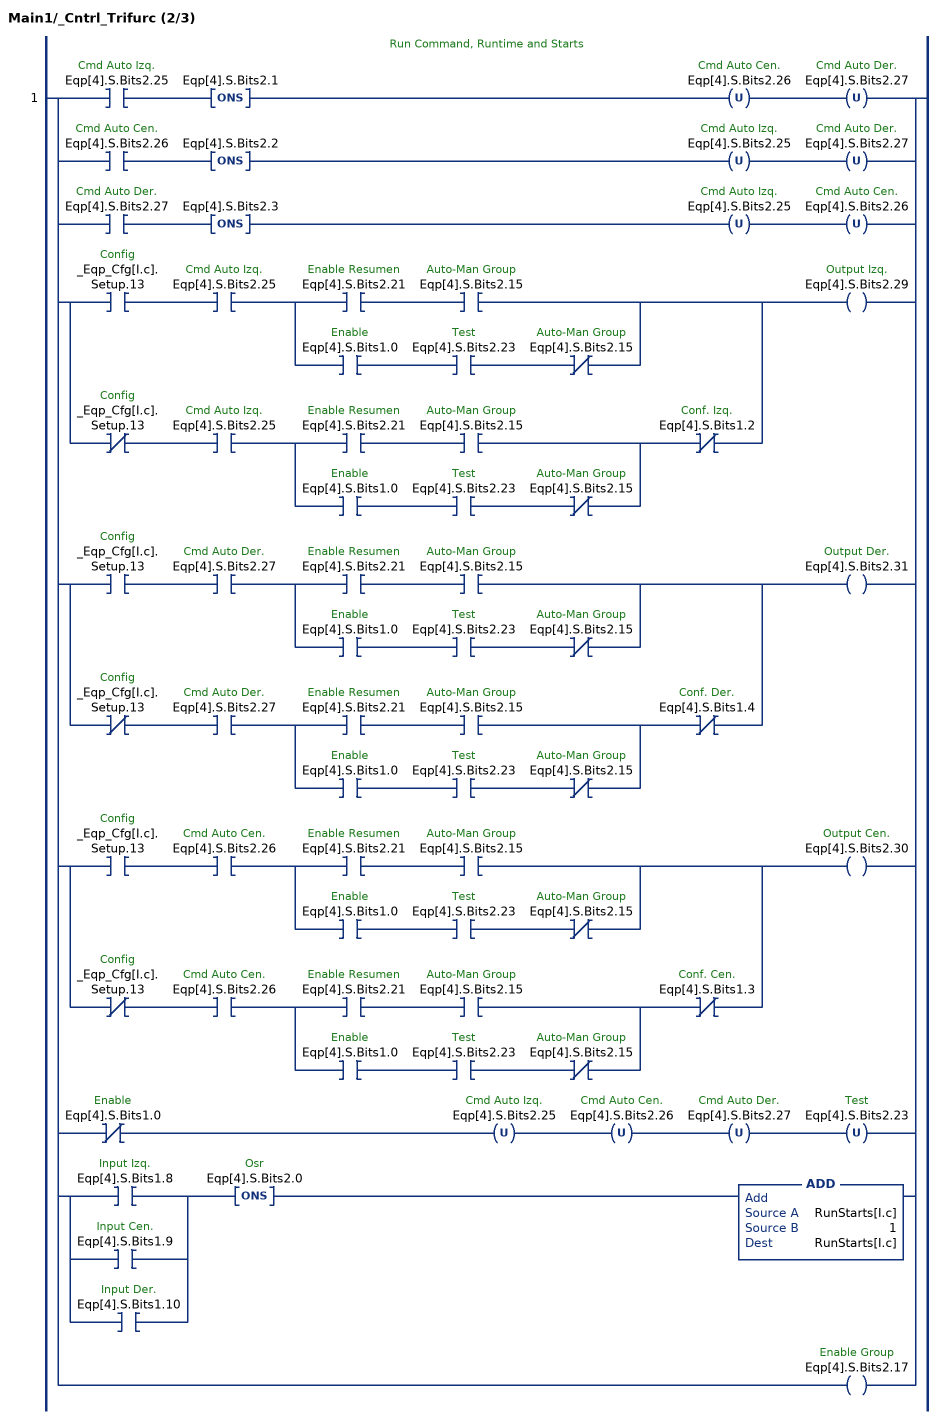
   // Run Command, Runtime and Starts
   1: [[XIC(Eqp[4].S.Bits2.25) ONS(Eqp[4].S.Bits2.1) OTU(Eqp[4].S.Bits2.26) OTU(Eqp[4].S.Bits2.27) ,XIC(Eqp[4].S.Bits2.26) ONS(Eqp[4].S.Bits2.2) OTU(Eqp[4].S.Bits2.25) OTU(Eqp[4].S.Bits2.27) ,XIC(Eqp[4].S.Bits2.27) ONS(Eqp[4].S.Bits2.3) OTU(Eqp[4].S.Bits2.25) OTU(Eqp[4].S.Bits2.26) ] ,[XIC(_Eqp_Cfg[I.c].Setup.13) XIC(Eqp[4].S.Bits2.25) [XIC(Eqp[4].S.Bits2.21) XIC(Eqp[4].S.Bits2.15) ,XIC(Eqp[4].S.Bits1.0) XIC(Eqp[4].S.Bits2.23) XIO(Eqp[4].S.Bits2.15) ] ,XIO(_Eqp_Cfg[I.c].Setup.13) XIC(Eqp[4].S.Bits2.25) [XIC(Eqp[4].S.Bits2.21) XIC(Eqp[4].S.Bits2.15) ,XIC(Eqp[4].S.Bits1.0) XIC(Eqp[4].S.Bits2.23) XIO(Eqp[4].S.Bits2.15) ] XIO(Eqp[4].S.Bits1.2) ] OTE(Eqp[4].S.Bits2.29) ,[XIC(_Eqp_Cfg[I.c].Setup.13) XIC(Eqp[4].S.Bits2.27) [XIC(Eqp[4].S.Bits2.21) XIC(Eqp[4].S.Bits2.15) ,XIC(Eqp[4].S.Bits1.0) XIC(Eqp[4].S.Bits2.23) XIO(Eqp[4].S.Bits2.15) ] ,XIO(_Eqp_Cfg[I.c].Setup.13) XIC(Eqp[4].S.Bits2.27) [XIC(Eqp[4].S.Bits2.21) XIC(Eqp[4].S.Bits2.15) ,XIC(Eqp[4].S.Bits1.0) XIC(Eqp[4].S.Bits2.23) XIO(Eqp[4].S.Bits2.15) ] XIO(Eqp[4].S.Bits1.4) ] OTE(Eqp[4].S.Bits2.31) ,[XIC(_Eqp_Cfg[I.c].Setup.13) XIC(Eqp[4].S.Bits2.26) [XIC(Eqp[4].S.Bits2.21) XIC(Eqp[4].S.Bits2.15) ,XIC(Eqp[4].S.Bits1.0) XIC(Eqp[4].S.Bits2.23) XIO(Eqp[4].S.Bits2.15) ] ,XIO(_Eqp_Cfg[I.c].Setup.13) XIC(Eqp[4].S.Bits2.26) [XIC(Eqp[4].S.Bits2.21) XIC(Eqp[4].S.Bits2.15) ,XIC(Eqp[4].S.Bits1.0) XIC(Eqp[4].S.Bits2.23) XIO(Eqp[4].S.Bits2.15) ] XIO(Eqp[4].S.Bits1.3) ] OTE(Eqp[4].S.Bits2.30) ,XIO(Eqp[4].S.Bits1.0) OTU(Eqp[4].S.Bits2.25) OTU(Eqp[4].S.Bits2.26) OTU(Eqp[4].S.Bits2.27) OTU(Eqp[4].S.Bits2.23) ,[XIC(Eqp[4].S.Bits1.8) ,XIC(Eqp[4].S.Bits1.9) ,XIC(Eqp[4].S.Bits1.10) ] ONS(Eqp[4].S.Bits2.0) ADD(RunStarts[I.c],1,RunStarts[I.c]) ,OTE(Eqp[4].S.Bits2.17) ];
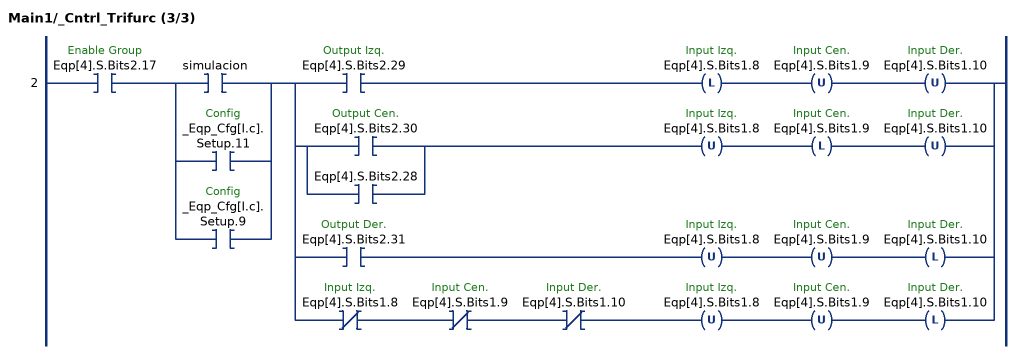
   2: XIC(Eqp[4].S.Bits2.17)[XIC(simulacion) ,XIC(_Eqp_Cfg[I.c].Setup.11) ,XIC(_Eqp_Cfg[I.c].Setup.9) ][XIC(Eqp[4].S.Bits2.29) OTL(Eqp[4].S.Bits1.8) OTU(Eqp[4].S.Bits1.9) OTU(Eqp[4].S.Bits1.10) ,[XIC(Eqp[4].S.Bits2.30) ,XIC(Eqp[4].S.Bits2.28) ] OTU(Eqp[4].S.Bits1.8) OTL(Eqp[4].S.Bits1.9) OTU(Eqp[4].S.Bits1.10) ,XIC(Eqp[4].S.Bits2.31) OTU(Eqp[4].S.Bits1.8) OTU(Eqp[4].S.Bits1.9) OTL(Eqp[4].S.Bits1.10) ,XIO(Eqp[4].S.Bits1.8) XIO(Eqp[4].S.Bits1.9) XIO(Eqp[4].S.Bits1.10) OTU(Eqp[4].S.Bits1.8) OTU(Eqp[4].S.Bits1.9) OTL(Eqp[4].S.Bits1.10) ];
END_ROUTINE
